// TIA Portal V19 export
DATA_BLOCK "BUFFER"   // DB26
{ S7_Optimized_Access := 'FALSE' }
   VAR
      HMI_START : Bool;
      HMI_STOP : Bool;
      "MODE SELECTION" : Int;
      PROCESS : Int;
      Static_1 : Int;
      HMI_AUTO : Bool;
      HMI_MANUAL : Bool;
      HMI_STANDBY : Bool;
      "RECIPE DOWNLOAD" : Bool;
      "LEVEL BUFFER SWT" : Int;
      "LEVEL BUFFER PWT" : Int;
      "RINSE-1" : Int;
      "ACID / ALAKLI" : Int;
      "RINSE-2" : Int;
      "RINSE-3" : Int;
      FINAL_RINSE : Int;
      CONTINUE : Bool;
      RESET : Bool;
      phMAINTAIN : Bool;
   END_VAR
BEGIN
END_DATA_BLOCK
